TYPE ST_variables :
STRUCT
	bEnable   : BOOL;
    bStop     : BOOL;
    bMoveRel  : BOOL;
    rVelocity : REAL;
    rDistance : REAL;
END_STRUCT
END_TYPE

(* stored: Version 1.1.0.1, ProductVersion 3.1.4024.16
   DUT ST_variables: Id {420a4d57-bd22-4386-a464-55b704e4b2c4} *)
